FUNCTION_BLOCK DoorModel
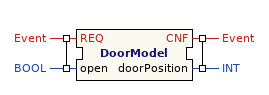
  EVENT_INPUT
    REQ WITH open;
  END_EVENT
  EVENT_OUTPUT
    CNF WITH doorPosition;
  END_EVENT
  VAR_INPUT
    open : BOOL;
  END_VAR
  VAR_OUTPUT
    doorPosition : INT;
  END_VAR
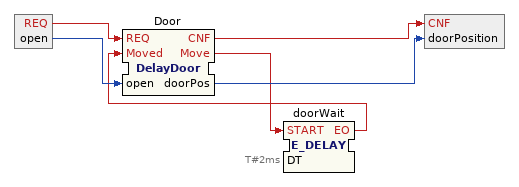
  FBS
    doorWait : E_DELAY(DT := T#2ms);
    Door : DelayDoor;
  END_FBS
  EVENT_CONNECTIONS
    REQ TO Door.REQ;
    doorWait.EO TO Door.Moved;
    Door.CNF TO CNF;
    Door.Move TO doorWait.START;
  END_CONNECTIONS
  DATA_CONNECTIONS
    open TO Door.open;
    Door.doorPos TO doorPosition;
  END_CONNECTIONS
END_FUNCTION_BLOCK
